(* IEC 61131-3 sources: Industry-PLC-LLM/data/PLCBEAD_repo/PLCBEAD_PLCEmbed-main/PLC-BEAD/Source/GEB/_BYTE_TO_REAL, 1 file *)

(* ---- _BYTE_TO_REAL.ST ---- *)
FUNCTION _BYTE_TO_REAL:REAL
	VAR_INPUT
		IN :	BYTE;
	END_VAR

	_BYTE_TO_REAL := USINT_TO_REAL(BYTE_TO_USINT(IN));
END_FUNCTION

PROGRAM program0
  VAR
    LocalVar0 : BYTE;
	LocalOUT  : REAL;
  END_VAR

  LocalOUT := _BYTE_TO_REAL(LocalVar0);
END_PROGRAM
